TYPE ST_PneumaticAxisFBConfig :
STRUCT
    nTimeToExtend: INT; //User defined time for the cylider to extract in seconds
    nTimeToRetract: INT; //User defined time for the cylinder to retract in seconds
    nTimeElapsedExtend: INT; //Elapsed time while extracting cylinder
    nTimeElapsedRetract: INT; //Elapsed time while retracting cylinder
END_STRUCT
END_TYPE

(* stored: Version 1.1.0.1, ProductVersion 3.1.4024.5
   DUT ST_PneumaticAxisFBConfig: Id {0cf5a73f-3f7b-4191-a68d-fd09f581360b} *)
